FUNCTION_BLOCK FB_BlinkingLight
VAR_INPUT
	dwTimeOn : DWORD;
	dwTimeOff : DWORD;
END_VAR
VAR_OUTPUT
	bLight : BOOL;	// Determines whether the light will be ON or OFF
END_VAR
VAR
	fbTimerOn : TON;
	fbTimerOff : TON;
	fbStartTrigger : R_TRIG;
	
	nCurrentPhase : INT := 10;	// 10 - ON, 20 - OFF
	
	bIsBlinking : bool;
END_VAR

CASE nCurrentPhase OF
    10:	// ON
        fbTimerOn(IN := TRUE, PT := DWORD_TO_TIME(dwTimeOn));
        IF fbTimerOn.Q THEN
            fbTimerOn(IN := FALSE); // Reset the on timer
            nCurrentPhase := 20;  // Move to the off phase
        END_IF
        bLight := TRUE;

    20:	// OFF
        fbTimerOff(IN := TRUE, PT := DWORD_TO_TIME(dwTimeOff));
        IF fbTimerOff.Q THEN
            fbTimerOff(IN := FALSE); // Reset the off timer
            nCurrentPhase := 10;  // Move to the On phase
        END_IF
        bLight := FALSE;
		
ELSE
	fbTimerOn(IN := FALSE);
    fbTimerOff(IN := FALSE);
    bLight := FALSE;
END_CASE

END_FUNCTION_BLOCK

(* stored: Version 1.1.0.1, ProductVersion 3.1.4024.12
   POU FB_BlinkingLight: Id {dc350849-3efc-47f9-a2a8-3b706b4b516e}, SpecialFunc None *)
